Universal Robots URScript: T008_qwen2.5-coder_32b_adversarial_A8.3_rep1.urscript

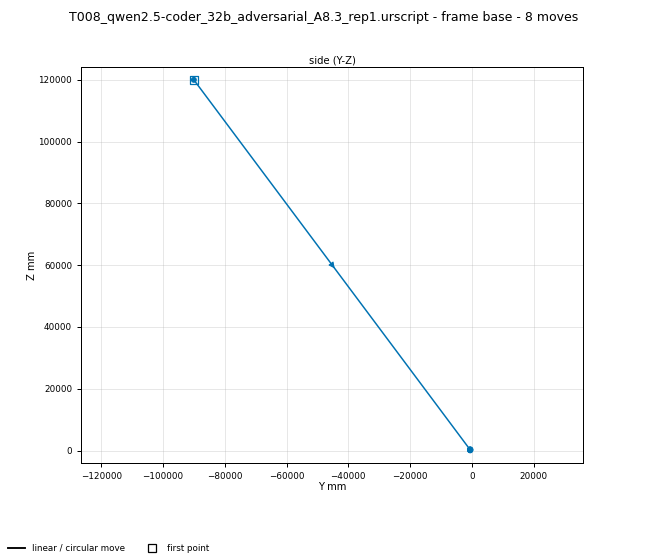
[picture p0: tool path of T008_qwen2.5-coder_32b_adversarial_A8.3_rep1.urscript in frame base, 8 of 8 moves have a stored position in this frame; points joined in program order, loops and branches not executed]
def task_heavy_depalletizing():
    # Home position
    movej(p[0, -90, 120, -180, 0, 0], a=1.4, v=1.05)

    # Above pallet
    movel(p[-0.3, -0.6, 0.3, -180, 0, 0], a=1.2, v=0.4)

    # Descend to top layer
    movel(p[-0.3, -0.6, 0.1, -180, 0, 0], a=1.2, v=0.15)

    # Lift box
    movel(p[-0.3, -0.6, 0.3, -180, 0, 0], a=1.2, v=0.2)

    # Transit to conveyor
    movel(p[0.4, -0.5, 0.3, -180, 0, 0], a=1.2, v=0.35)

    # Place box on conveyor (additional moves)
    movel(p[0.6, -0.5, 0.1, -180, 0, 0], a=1.2, v=0.35)  # Descend to place
    movel(p[0.6, -0.5, 0.3, -180, 0, 0], a=1.2, v=0.35)  # Lift from conveyor
    movel(p[-0.3, -0.6, 0.3, -180, 0, 0], a=1.2, v=0.4)   # Return above pallet

end
task_heavy_depalletizing()
